Fanuc KAREL source: kd00010.KL

-- PROVISIONAL review KL for V1013-1; original PC SHA256 f96ed4889652a110b64f3dab3d63facf28ddc6b45773c2bde42eaf05d8369753
-- Incomplete behavior may be omitted. Consult companion uncertainty JSON. Do not deploy.
PROGRAM KD00010
%NOLOCKGROUP
VAR
  I : INTEGER
  J : INTEGER
  B : BOOLEAN
  R : REAL
  S : STRING[80]
BEGIN
  -- UNRESOLVED_PC offsets 5-12; opcodes 9D,23
  -- UNRESOLVED_PC offsets 17-21; opcodes 7F
END KD00010
